FUNCTION_BLOCK WeightSensor IMPLEMENTS ITF_AnalogSensor
VAR_INPUT
END_VAR
VAR_OUTPUT
END_VAR
VAR
	AI_WPWeight AT %I* : INT;
END_VAR

PROPERTY Value : INT
GET
Value := AI_WPWeight;
END_GET
END_PROPERTY

END_FUNCTION_BLOCK

(* stored: Version 1.1.0.1, ProductVersion 3.1.4024.9
   POU WeightSensor: Id {a5cdfec8-362e-441f-b9b1-ba6103586d0f}, SpecialFunc None
   Property Value: Id {5b504a1f-3cfe-4daa-b35c-2c2a13a0655b}
   Get Get: Id {6887616e-82f1-47e0-a49c-207d10de3c31} *)
